FUNCTION_BLOCK FB_BaseGroupElementDecoratorParent EXTENDS FB_BaseControlElementDecoratorParent IMPLEMENTS ITF_BaseGroupElementDecoratorParent
VAR
	itfGroupElement				: ITF_BaseGroupElement;
END_VAR

(*			
	EVERDE sp. z o.o.
	Rafał Osajda		24.03.2025		TC 4024.66
	Definicja nowego zgłoszenia
*)
METHOD PUBLIC EventsDefinition : BOOL
EventsDefinition		:= THIS^.itfGroupElement.EventsDefinition ();
END_METHOD

(*			
	EVERDE sp. z o.o.
	Rafał Osajda		27.03.2025		TC 4024.66
	Obsluga bledow sprawdzanie czy jakis blad sie nei pojawil i ustawienie stanu lub wylaczenie
*)
METHOD PUBLIC ExecuteEveryCycle_Error
VAR_INPUT
END_VAR
THIS^.itfGroupElement.ExecuteEveryCycle_Error ();
END_METHOD

(*			
	EVERDE sp. z o.o.
	Rafał Osajda		27.03.2025		TC 4024.66
	Wywolanie co cykl operacji 
*)
METHOD PUBLIC ExecuteEveryCycle_Operation
VAR_INPUT
END_VAR
THIS^.itfGroupElement.ExecuteEveryCycle_Operation ();
END_METHOD

(*			
	EVERDE sp. z o.o.
	Rafał Osajda		27.03.2025		TC 4024.66
	Aktualizacja flag 
*)
METHOD PUBLIC ExecuteEveryCycle_Status
VAR_INST
END_VAR
THIS^.itfGroupElement.ExecuteEveryCycle_Status ();
END_METHOD

(*			
	EVERDE sp. z o.o.
	Rafał Osajda		27.03.2025		TC 4024.66
	Testowanie czy nei pojawil sie jakis rozkaz i uruchomienie odpowiednich operacji
*)
METHOD PUBLIC ExecuteEveryCycle_Test
VAR_INPUT
END_VAR
THIS^.itfGroupElement.ExecuteEveryCycle_Test ();
END_METHOD

METHOD FB_init : BOOL
VAR_INPUT
	bInitRetains : BOOL; // if TRUE, the retain variables are initialized (warm start / cold start)
	bInCopyCode : BOOL;  // if TRUE, the instance afterwards gets moved into the copy code (online change)
	fbToDecorate		: ITF_DecoratedElement;
END_VAR
THIS^.itfGroupElement	:= fbToDecorate.GetITFGroupElement ();
END_METHOD

(*			
	EVERDE sp. z o.o.
	Rafał Osajda		03.10.2025		TC 4024.66
	
*)
METHOD PUBLIC FirstCycle : BOOL
VAR_INPUT
END_VAR
FirstCycle				:= THIS^.itfGroupElement.FirstCycle ();
END_METHOD

METHOD PUBLIC GetCode : STRING
VAR_INPUT
END_VAR
GetCode			:= THIS^.itfGroupElement.GetCode ();
END_METHOD

(*			
	EVERDE sp. z o.o.
	Rafał Osajda		30.04.2025		TC 4024.66
	Zwraca czy element jest czymś zajety
*)
METHOD PUBLIC GetDoNothing : BOOL
GetDoNothing		:= THIS^.itfGroupElement.GetDoNothing ();
END_METHOD

METHOD PUBLIC GetID : UINT
VAR_INPUT
END_VAR
GetID		:= THIS^.itfGroupElement.GetID ();
END_METHOD

METHOD PUBLIC GetIdentyfier : ST_BaseElementIdentifier
VAR_INPUT
END_VAR
GetIdentyfier		:= THIS^.itfGroupElement.GetIdentyfier ();
END_METHOD

METHOD PUBLIC GetName : ST_BaseLabel
VAR_INPUT
END_VAR
GetName		:= THIS^.itfGroupElement.GetName ();
END_METHOD

(*			
	EVERDE sp. z o.o.
	Rafał Osajda		30.04.2025		TC 4024.66
	Zwraca czy element jest w pozycji 0 - referencyjnej
*)
METHOD PUBLIC GetPosition0 : BOOL
GetPosition0	:= THIS^.itfGroupElement.GetPosition0 ();
END_METHOD

METHOD PUBLIC GetType : E_BaseElementType
VAR_INPUT
END_VAR
GetType		:= THIS^.itfGroupElement.GetType ();
END_METHOD

(*			
	EVERDE sp. z o.o.
	Rafał Osajda		31.03.2025		TC 4024.66
	Flaga że w tej sesji pracy maszyny element został już wybazowany
*)
METHOD PUBLIC HomingGetDone : BOOL
VAR_INPUT
END_VAR
HomingGetDone	:= THIS^.itfGroupElement.HomingGetDone ();
END_METHOD

(*			
	EVERDE sp. z o.o.
	Rafał Osajda		11.04.2025		TC 4024.66
	Zwraca czy bazowanie jest potrzebne
*)
METHOD PUBLIC HomingGetIsNeeded : BOOL
VAR_INPUT
END_VAR
HomingGetIsNeeded	:= THIS^.itfGroupElement.HomingGetIsNeeded ();
END_METHOD

(*			
	EVERDE sp. z o.o.
	Rafał Osajda		27.05.2025		TC 4024.66
	Uruchomienie metody bazowania
*)
METHOD PUBLIC HomingStart
VAR_INPUT
END_VAR
THIS^.itfGroupElement.HomingStart ();
END_METHOD

METHOD PUBLIC IsValidCommonData : BOOL
VAR_INPUT
END_VAR
IsValidCommonData			:= THIS^.itfGroupElement.IsValidCommonData ();
END_METHOD

(*			
	EVERDE sp. z o.o.
	Rafał Osajda		07.10.2025		TC 4024.66
	Dodpisywanie się do listy logera
*)
METHOD PUBLIC JoinTheLogger : BOOL
VAR_INPUT
END_VAR
JoinTheLogger	:= THIS^.itfGroupElement.JoinTheLogger ();
END_METHOD

METHOD PUBLIC LinkCommonData : BOOL
VAR_INPUT
	stCommonData				: REFERENCE TO ST_BaseCommonData;
END_VAR
LinkCommonData			:= THIS^.itfGroupElement.LinkCommonData (stCommonData := stCommonData);
END_METHOD

METHOD PUBLIC LinkSS1 : BOOL
VAR_INPUT
	fbSS1			: ITF_BaseFlagGet;
END_VAR
LinkSS1		:= THIS^.itfGroupElement.LinkSS1 (fbSS1 := fbSS1);
END_METHOD

METHOD PUBLIC LinkSTO : BOOL
VAR_INPUT
	fbSTO			: ITF_BaseFlagGet;
END_VAR
LinkSTO		:= THIS^.itfGroupElement.LinkSTO (fbSTO := fbSTO);
END_METHOD

(*			
	EVERDE sp. z o.o.
	Rafał Osajda		31.03.2025		TC 4024.66
	Zwraca status zasilania	
*)
METHOD PUBLIC PowerGetStatus : BOOL
VAR_INPUT
END_VAR
PowerGetStatus		:= THIS^.itfGroupElement.PowerGetStatus ();
END_METHOD

(*			
	EVERDE sp. z o.o.
	Rafał Osajda		31.03.2025		TC 4024.66
	Wyłączenie zasilania
*)
METHOD PUBLIC PowerTurnOff : BOOL
VAR_INPUT
END_VAR
PowerTurnOff		:= THIS^.itfGroupElement.PowerTurnOff ();
END_METHOD

(*			
	EVERDE sp. z o.o.
	Rafał Osajda		31.03.2025		TC 4024.66
	Uruchomienie zasialania
*)
METHOD PUBLIC PowerTurnOn
VAR_INPUT
END_VAR
THIS^.itfGroupElement.PowerTurnOn ();
END_METHOD

METHOD PUBLIC Reset : BOOL
VAR_INPUT
END_VAR
Reset	:= THIS^.itfGroupElement.Reset ();
END_METHOD

METHOD PUBLIC ResetGetBusy : BOOL
VAR_INPUT
END_VAR
ResetGetBusy		:= THIS^.itfGroupElement.ResetGetBusy ();
END_METHOD

METHOD PUBLIC ResetGetStatus : BOOL
VAR_INPUT
END_VAR
ResetGetStatus			:= THIS^.itfGroupElement.ResetGetStatus ();
END_METHOD

METHOD PUBLIC SetCode
VAR_INPUT
	sCode							: STRING;
	sAdd							: STRING;
END_VAR
THIS^.itfGroupElement.SetCode (sCode := sCode, sAdd := sAdd);
END_METHOD

(*			
	EVERDE sp. z o.o.
	Rafał Osajda		03.10.2025		TC 4024.66
	nadawanie unikalnych ID dla zdarzeń
*)
METHOD PUBLIC SetEventsIDs : UINT
VAR_INPUT
	uiNewID		: UINT;
END_VAR
SetEventsIDs		:= THIS^.itfGroupElement.SetEventsIDs (uiNewID := uiNewID);
END_METHOD

METHOD PUBLIC SetID : UINT
VAR_INPUT
	uiID					: UINT;
END_VAR
SetID		:= THIS^.itfGroupElement.SetID (uiID := uiID);
END_METHOD

METHOD PUBLIC SetName
VAR_INPUT
	stName				: ST_BaseLabel;
END_VAR
THIS^.itfGroupElement.SetName (stName := stName);
END_METHOD

METHOD PUBLIC SetType
VAR_INPUT
	eType					: E_BaseElementType;
END_VAR
THIS^.itfGroupElement.SetType (eType := eType);
END_METHOD

END_FUNCTION_BLOCK

(* stored: Version 1.1.0.1
   POU FB_BaseGroupElementDecoratorParent: Id {7314ca7f-9a71-0330-3cec-f7962be5af3f}, SpecialFunc None
   Folder Bazowanie: Id {85b8fb0b-ab31-02a1-2a6a-5218858a76e4}
   Folder Events: Id {e8351569-4cac-0552-3608-afbacc7e4230}
   Folder ID: Id {4edcc3ce-685c-0bdb-20ad-18f1093ac4e3}
   Folder ITF_BaseComponent: Id {25e1184d-4b36-0512-1cc6-ef400d11f666}
   Folder WiazanieZmiennych: Id {746193b2-40d7-0f47-2f0c-6d00f6a5c71d}
   Folder Zasilanie: Id {05b58235-938c-0558-3e2a-af4cbe4f20a3}
   Method EventsDefinition: Id {e23e6e98-dcbd-061b-3ff7-b5caf5358e00}
   Method ExecuteEveryCycle_Error: Id {5f158b9f-40b1-0c42-31f9-163420752a8d}
   Method ExecuteEveryCycle_Operation: Id {dac4054b-33a7-0e2f-0220-003d3517c04a}
   Method ExecuteEveryCycle_Status: Id {d99e2865-581f-0821-38bb-7f091299311f}
   Method ExecuteEveryCycle_Test: Id {ad832635-2127-0d4c-3a51-f7d02ecb4e18}
   Method FB_init: Id {a4e33f86-77a8-0005-2645-34f0be7aeb52}
   Method FirstCycle: Id {d5ec58ec-8f16-07f2-0459-f26fc0936a9e}
   Method GetCode: Id {05ac98ee-2999-0fc8-15f6-68716ba17bca}
   Method GetDoNothing: Id {be2e6d5e-5419-0373-2ae1-dfe1d748d141}
   Method GetID: Id {fc482f15-e7db-0733-19ef-d6efc3a313e2}
   Method GetIdentyfier: Id {849bf7f9-1595-0275-1493-53577d7674db}
   Method GetName: Id {8853e2a5-c089-018f-2b3a-1e81625626d5}
   Method GetPosition0: Id {379a403c-af17-0aaa-017a-f47b998d0957}
   Method GetType: Id {7015a4e6-290c-060f-2833-4d1d91b16d41}
   Method HomingGetDone: Id {c1379eb4-bb57-0e51-0080-82ff53ee4fb6}
   Method HomingGetIsNeeded: Id {f8bea682-8c30-0a57-321b-e2e84c6a58ad}
   Method HomingStart: Id {fe11a7c5-f712-090d-1023-7a7ad33bd099}
   Method IsValidCommonData: Id {99461ccc-bd2c-0400-1c75-64cba24b7b1c}
   Method JoinTheLogger: Id {8ce1ac7b-2aec-0e14-2af1-ba22382210d1}
   Method LinkCommonData: Id {2d53e34f-01b8-048a-2b11-a6b1a6ec8474}
   Method LinkSS1: Id {bf34ea97-5a49-0254-0e58-426eb250b020}
   Method LinkSTO: Id {05d1e742-565b-0308-2851-95f2b965a2d7}
   Method PowerGetStatus: Id {108f43d4-51ba-0b13-188c-24862c57dc84}
   Method PowerTurnOff: Id {f3884bb7-c11e-07d6-04d0-fd5a789833a6}
   Method PowerTurnOn: Id {e2578f76-b9b3-0659-12cc-88e513220a63}
   Method Reset: Id {9eb124f0-a152-092b-08fe-798e3c29e95b}
   Method ResetGetBusy: Id {594902f7-c854-0e5d-2d56-e9d793912f08}
   Method ResetGetStatus: Id {a1d0aed7-0143-030a-0673-814c850837a6}
   Method SetCode: Id {21774ac8-6074-0cca-00e9-097c0fbb27b6}
   Method SetEventsIDs: Id {5d5c0813-46d6-0d65-0e64-fb332ca4d9c8}
   Method SetID: Id {fcd29c43-7f9a-0490-0225-f7f1b6c96306}
   Method SetName: Id {b820f42b-c477-0f04-1a2e-b37d2e6b8e9a}
   Method SetType: Id {aa8cd11a-6f0d-0b68-3941-67deaf4d7f91} *)
